// LS Electric XG5000 project: 8_23
// PLC LSPLC
// module base 0 slot 0: 입출력 모듈:XBC-DR14E (DC 24V 입력 8점, 릴레이 출력 6점)

PROGRAM NewProgram (task: 스캔 프로그램)

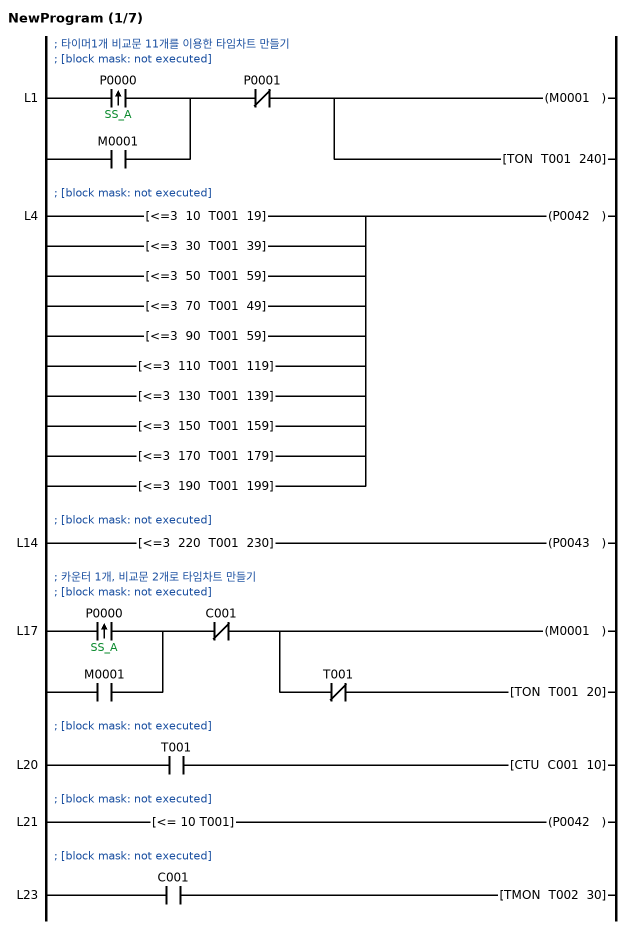
// 타이머1개 비교문 11개를 이용한 타임차트 만들기
; L1 (block mask: not executed)
LOADP     P0000	// SS_A
OR        M0001
AND NOT   P0001
OUT       M0001
TON       T001 240
; L4 (block mask: not executed)
LOAD<=3   10 T001 19
OR<=3     30 T001 39
OR<=3     50 T001 59
OR<=3     70 T001 49
OR<=3     90 T001 59
OR<=3     110 T001 119
OR<=3     130 T001 139
OR<=3     150 T001 159
OR<=3     170 T001 179
OR<=3     190 T001 199
OUT       P0042
; L14 (block mask: not executed)
LOAD<=3   220 T001 230
OUT       P0043
// 카운터 1개, 비교문 2개로 타임차트 만들기
; L17 (block mask: not executed)
LOADP     P0000	// SS_A
OR        M0001
AND NOT   C001
OUT       M0001
AND NOT   T001
TON       T001 20
; L20 (block mask: not executed)
LOAD      T001
CTU       C001 10
; L21 (block mask: not executed)
LOAD<=    10 T001
OUT       P0042
; L23 (block mask: not executed)
LOAD      C001
TMON      T002 30

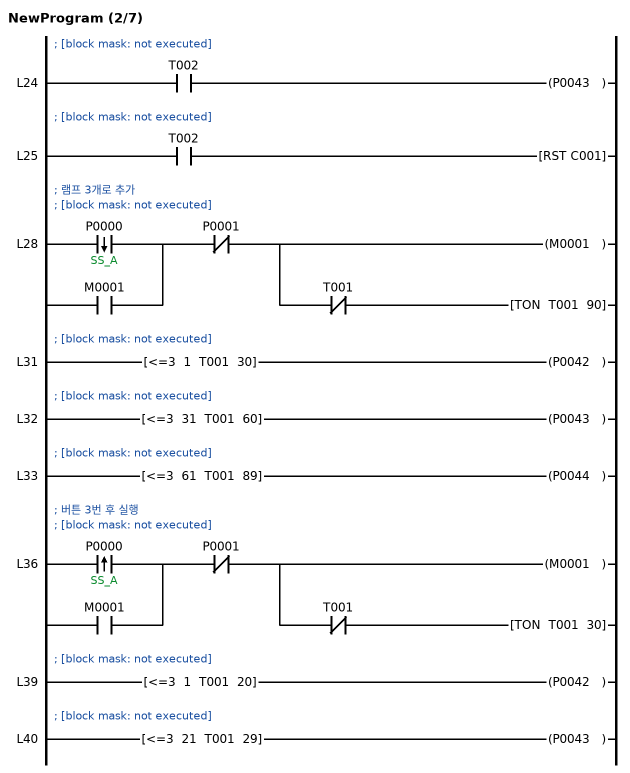
; L24 (block mask: not executed)
LOAD      T002
OUT       P0043
; L25 (block mask: not executed)
LOAD      T002
RST       C001
// 램프 3개로 추가
; L28 (block mask: not executed)
LOADN     P0000	// SS_A
OR        M0001
AND NOT   P0001
OUT       M0001
AND NOT   T001
TON       T001 90
; L31 (block mask: not executed)
LOAD<=3   1 T001 30
OUT       P0042
; L32 (block mask: not executed)
LOAD<=3   31 T001 60
OUT       P0043
; L33 (block mask: not executed)
LOAD<=3   61 T001 89
OUT       P0044
// 버튼 3번 후 실행
; L36 (block mask: not executed)
LOADP     P0000	// SS_A
OR        M0001
AND NOT   P0001
OUT       M0001
AND NOT   T001
TON       T001 30
; L39 (block mask: not executed)
LOAD<=3   1 T001 20
OUT       P0042
; L40 (block mask: not executed)
LOAD<=3   21 T001 29
OUT       P0043

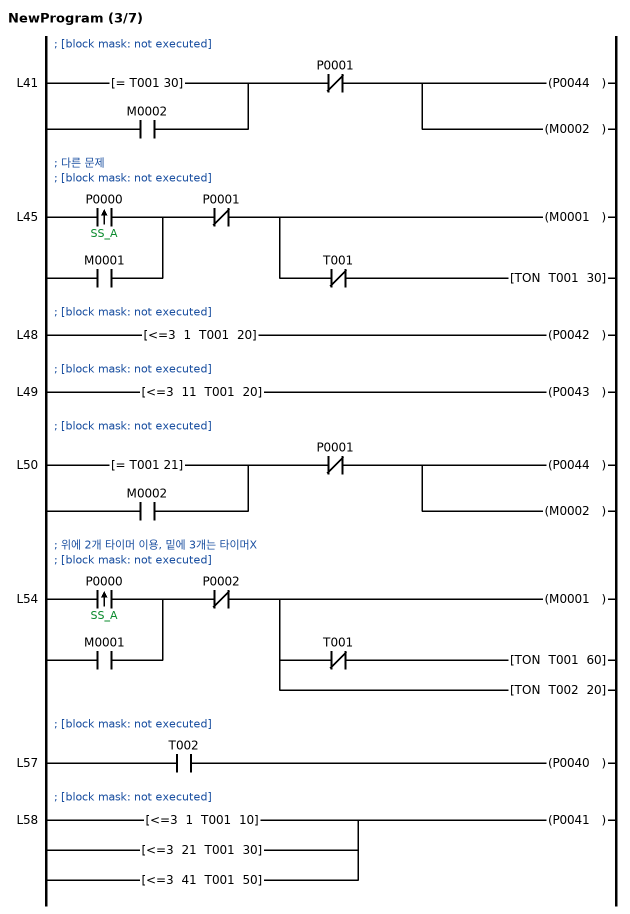
; L41 (block mask: not executed)
LOAD=     T001 30
OR        M0002
AND NOT   P0001
OUT       P0044
OUT       M0002
// 다른 문제
; L45 (block mask: not executed)
LOADP     P0000	// SS_A
OR        M0001
AND NOT   P0001
OUT       M0001
AND NOT   T001
TON       T001 30
; L48 (block mask: not executed)
LOAD<=3   1 T001 20
OUT       P0042
; L49 (block mask: not executed)
LOAD<=3   11 T001 20
OUT       P0043
; L50 (block mask: not executed)
LOAD=     T001 21
OR        M0002
AND NOT   P0001
OUT       P0044
OUT       M0002
// 위에 2개 타이머 이용, 밑에 3개는 타이머X
; L54 (block mask: not executed)
LOADP     P0000	// SS_A
OR        M0001
AND NOT   P0002
OUT       M0001
MPUSH
AND NOT   T001
TON       T001 60
MPOP
TON       T002 20
; L57 (block mask: not executed)
LOAD      T002
OUT       P0040
; L58 (block mask: not executed)
LOAD<=3   1 T001 10
OR<=3     21 T001 30
OR<=3     41 T001 50
OUT       P0041

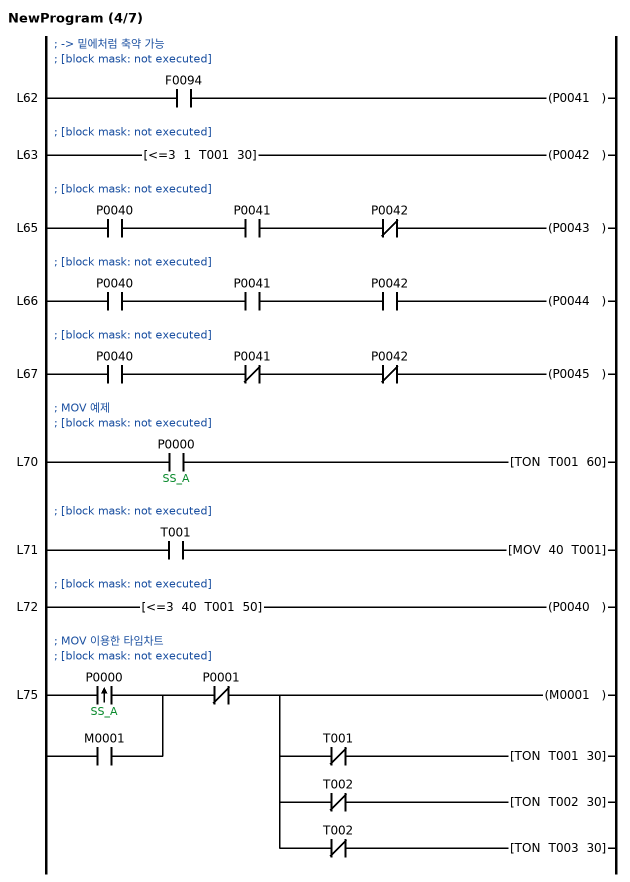
// -> 밑에처럼 축약 가능
; L62 (block mask: not executed)
LOAD      F0094
OUT       P0041
; L63 (block mask: not executed)
LOAD<=3   1 T001 30
OUT       P0042
; L65 (block mask: not executed)
LOAD      P0040
AND       P0041
AND NOT   P0042
OUT       P0043
; L66 (block mask: not executed)
LOAD      P0040
AND       P0041
AND       P0042
OUT       P0044
; L67 (block mask: not executed)
LOAD      P0040
AND NOT   P0041
AND NOT   P0042
OUT       P0045
// MOV 예제
; L70 (block mask: not executed)
LOAD      P0000	// SS_A
TON       T001 60
; L71 (block mask: not executed)
LOAD      T001
MOV       40 T001
; L72 (block mask: not executed)
LOAD<=3   40 T001 50
OUT       P0040
// MOV 이용한 타임차트
; L75 (block mask: not executed)
LOADP     P0000	// SS_A
OR        M0001
AND NOT   P0001
OUT       M0001
MPUSH
AND NOT   T001
TON       T001 30
MLOAD
AND NOT   T002
TON       T002 30
MPOP
AND NOT   T002
TON       T003 30

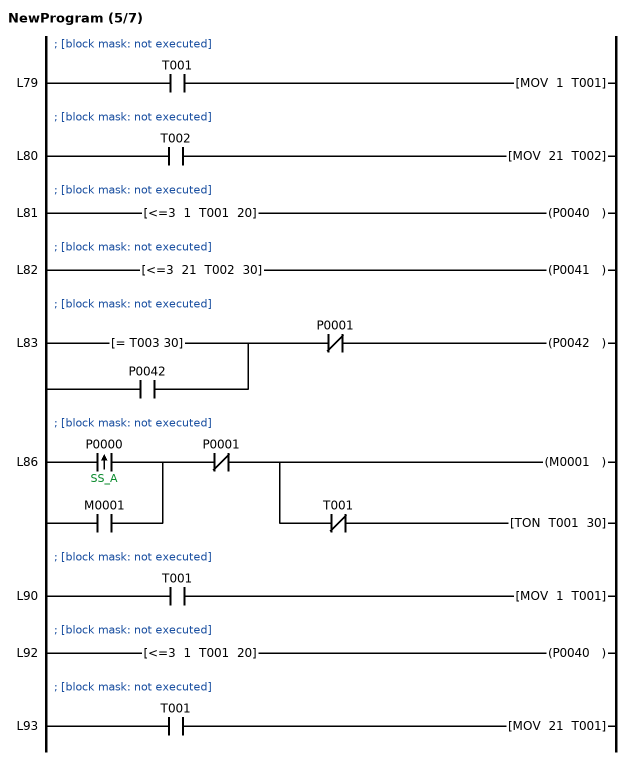
; L79 (block mask: not executed)
LOAD      T001
MOV       1 T001
; L80 (block mask: not executed)
LOAD      T002
MOV       21 T002
; L81 (block mask: not executed)
LOAD<=3   1 T001 20
OUT       P0040
; L82 (block mask: not executed)
LOAD<=3   21 T002 30
OUT       P0041
; L83 (block mask: not executed)
LOAD=     T003 30
OR        P0042
AND NOT   P0001
OUT       P0042
; L86 (block mask: not executed)
LOADP     P0000	// SS_A
OR        M0001
AND NOT   P0001
OUT       M0001
AND NOT   T001
TON       T001 30
; L90 (block mask: not executed)
LOAD      T001
MOV       1 T001
; L92 (block mask: not executed)
LOAD<=3   1 T001 20
OUT       P0040
; L93 (block mask: not executed)
LOAD      T001
MOV       21 T001

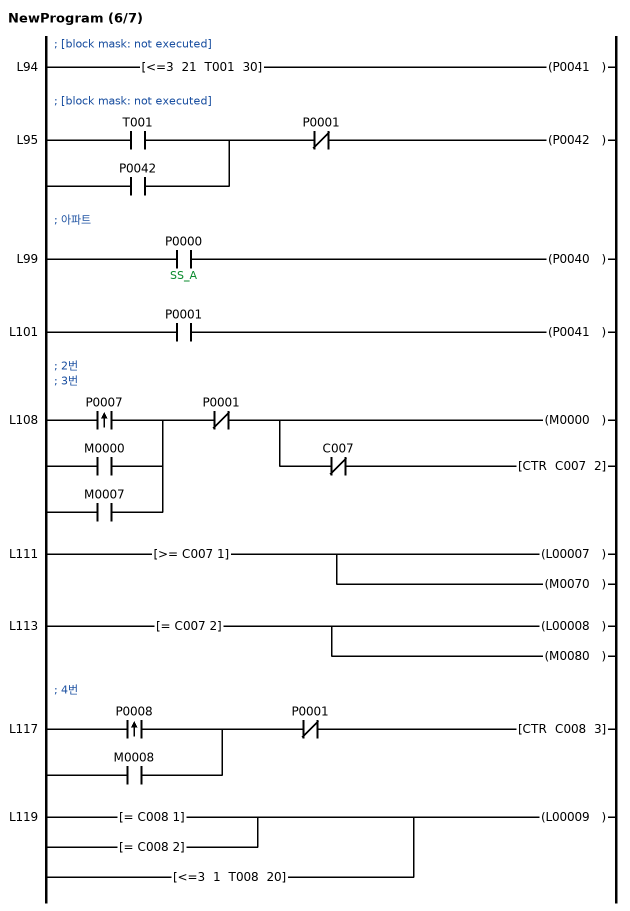
; L94 (block mask: not executed)
LOAD<=3   21 T001 30
OUT       P0041
; L95 (block mask: not executed)
LOAD      T001
OR        P0042
AND NOT   P0001
OUT       P0042
// 아파트
; L99
LOAD      P0000	// SS_A
OUT       P0040
; L101
LOAD      P0001
OUT       P0041
// 2번
// 3번
; L108
LOADP     P0007
OR        M0000
OR        M0007
AND NOT   P0001
OUT       M0000
AND NOT   C007
CTR       C007 2
; L111
LOAD>=    C007 1
OUT       L00007
OUT       M0070
; L113
LOAD=     C007 2
OUT       L00008
OUT       M0080
// 4번
; L117
LOADP     P0008
OR        M0008
AND NOT   P0001
CTR       C008 3
; L119
LOAD=     C008 1
OR=       C008 2
OR<=3     1 T008 20
OUT       L00009

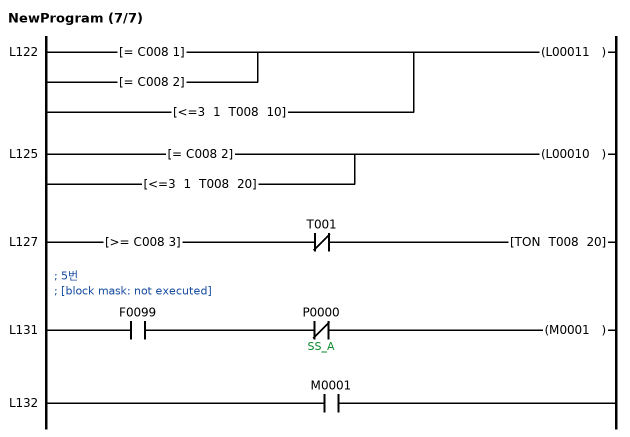
; L122
LOAD=     C008 1
OR=       C008 2
OR<=3     1 T008 10
OUT       L00011
; L125
LOAD=     C008 2
OR<=3     1 T008 20
OUT       L00010
; L127
LOAD>=    C008 3
AND NOT   T001
TON       T008 20
// 5번
; L131 (block mask: not executed)
LOAD      F0099
AND NOT   P0000	// SS_A
OUT       M0001
; L132
LOAD      M0001